FUNCTION_BLOCK FB_ControlSignal
VAR_INPUT
	fFF 			: LREAL;
	fPID			: LREAL;
	
	fDeadBandUp		: LREAL;
	fDeadBandDown	: LREAL;

	bPID			: BOOL;
	bFF				: BOOL;
	bU				: BOOL;
	bValve			: BOOL;
END_VAR
VAR_OUTPUT
	fU				: LREAL;
	fUAdj			: LREAL;
END_VAR
VAR
	FF				: LREAL;
	PID				: LREAL;
END_VAR


FF := fFF  * TO_INT(bFF);

PID := fPID * TO_INT(bPID);

fUAdj := (FF+PID)*TO_INT(bValve);

IF FF = 0.0 THEN
	fU := 0.0;
ELSE
	IF (fUAdj > 0.0) THEN
		fU := fUAdj + fDeadBandUp;
	ELSIF (fUAdj < 0.0) THEN
		fU := fUAdj - fDeadBandDown;
	ELSE
		fU := 0.0;
	END_IF
END_IF
IF fU < -1.0 THEN
	fU := -1.0;
ELSIF fU > 1.0 THEN
	fU := 1.0;
ELSE
	fU := fU;
END_IF

END_FUNCTION_BLOCK

(* stored: Version 1.1.0.1, ProductVersion 3.1.4024.12
   POU FB_ControlSignal: Id {5ec98e7b-f91c-4803-9df2-1eb6eb99ed16}, SpecialFunc None *)
